Yaskawa INFORM job: R1_W31(0,0)_KM-OK.JBI

/JOB
//NAME R1_W31(0,0)_KM-OK
///FOLDERNAME KRIS-SCIANA
//POS
///NPOS 65,65,0,4,0,0
///TOOL 0
///POSTYPE PULSE
///PULSE
C00000=-3378,-139883,-97046,148601,63097,19554
C00001=-9157,-139883,-97046,148601,63097,19554
C00002=14423,-139883,-97046,148601,63097,19554
C00003=25248,-128582,-94175,152681,55492,17228
C00004=27205,-127666,-93925,153637,54506,16635
C00005=25484,-128476,-94146,152795,55373,17157
C00006=24457,-124392,-93002,151737,54562,17917
C00007=25484,-128476,-94146,152795,55373,17157
C00008=16411,-139658,-96993,149510,62230,18973
C00009=16411,-139658,-96993,149510,62230,18973
C00010=23126,-128454,-94140,151543,56250,17966
C00011=25024,-127329,-93830,152407,55203,17428
C00012=26846,-126477,-93594,153294,54279,16874
C00013=25024,-127329,-93830,152407,55203,17428
C00014=24148,-123758,-92822,151495,54500,18086
C00015=22779,-128284,-94093,151343,56332,18098
C00016=21057,-113910,-69749,152741,63461,16563
C00017=22950,-111460,-69051,153499,62072,16185
C00018=24905,-111066,-68937,154492,61279,15593
C00019=26651,-110455,-68757,155377,60511,15074
C00020=24905,-111066,-68937,154492,61279,15593
C00021=24139,-108709,-68237,153879,60863,16039
C00022=24905,-111066,-68937,154492,61279,15593
C00023=21365,-129655,-79903,153341,64942,15994
C00024=21365,-129655,-79903,153341,64942,15994
C00025=21365,-129655,-79903,153341,64942,15994
C00026=20940,-133487,-97884,150530,57334,18616
C00027=26110,-127410,-97825,152085,52729,17755
///LIMIT ON
C00028=-107604,79582,41685,153491,37881,19627
C00029=-107224,79409,41473,153690,37712,19470
///LIMIT OFF
C00030=26036,-121266,-88084,153104,55194,16958
C00031=22153,-126078,-89436,151612,58043,17810
C00032=26151,-121055,-87868,153174,55168,16910
///LIMIT ON
C00033=-107258,82886,61095,119534,27741,31091
C00034=-106881,82684,60844,119663,27474,31013
///LIMIT OFF
C00035=26195,-120747,-87778,153163,55063,16923
C00036=26195,-120747,-87778,153163,55063,16923
C00037=27152,-120514,-87710,153662,54649,16609
///LIMIT ON
C00038=-107258,82806,60996,119500,27732,31108
C00039=-106881,82604,60746,119629,27464,31030
///LIMIT OFF
C00040=27152,-120514,-87710,153662,54649,16609
C00041=25896,-122880,-88390,153250,55792,16826
C00042=27161,-117906,-83715,154050,55615,16299
C00043=27161,-117906,-83715,154050,55615,16299
///LIMIT ON
C00044=-107257,82726,60897,119467,27722,31125
C00045=-106880,82524,60648,119596,27455,31047
///LIMIT OFF
C00046=27161,-117906,-83715,154050,55615,16299
C00047=26010,-116408,-78989,154106,57886,16118
C00048=26010,-116408,-78989,154106,57886,16118
C00049=27211,-114659,-78882,154502,56737,15929
///LIMIT ON
C00050=-107256,82646,60799,119433,27713,31142
C00051=-106879,82445,60550,119562,27446,31064
///LIMIT OFF
C00052=27209,-114651,-78879,154500,56735,15931
C00053=25407,-114144,-74093,154324,59707,15835
C00054=25407,-110889,-69044,154716,60962,15469
C00055=26831,-107525,-66907,155376,60119,15103
///LIMIT ON
C00056=-107256,82566,60701,119400,27704,31159
C00057=-106879,82365,60452,119529,27437,31081
///LIMIT OFF
C00058=27080,-101000,-56543,156267,62718,14289
C00059=22644,-108994,-60238,154325,65787,15230
C00060=-52788,-93244,-55241,130948,98095,35026
C00061=-80375,-99739,-69495,56806,86442,35710
C00062=-110141,-127728,-104321,3125,87796,34758
C00063=-110141,-127728,-104321,3125,87796,34758
C00064=1472,-127728,-104321,3125,87796,34758
BC00000=204370,1305091,673639
BC00001=2222,1298561,673639
BC00002=2222,1317543,673639
BC00003=2221,1317541,673640
BC00004=2221,1317541,673640
BC00005=2221,1317541,673640
BC00006=2221,1317541,673640
BC00007=2221,1317541,673640
BC00008=2221,1317541,673640
BC00009=2221,1317541,422792
BC00010=2221,1317541,422792
BC00011=2221,1317541,422792
BC00012=2221,1317541,422792
BC00013=2221,1317541,422792
BC00014=2221,1317541,422792
BC00015=2221,1317541,422792
BC00016=2221,1317541,335002
BC00017=2221,1317541,335002
BC00018=2221,1317541,335002
BC00019=2221,1317541,335002
BC00020=2221,1317541,335002
BC00021=2221,1317541,335002
BC00022=2221,1317541,335002
BC00023=2221,1317541,593632
BC00024=2221,1317541,809188
BC00025=12256,1314853,809188
BC00026=2183,1317396,719431
BC00027=2183,1317396,719431
BC00028=39399,1318630,622069
BC00029=39399,1318630,622069
BC00030=2183,1317396,719431
BC00031=2183,1317396,689296
BC00032=2183,1317396,649606
BC00033=22077,1294776,797041
BC00034=22077,1294776,797041
BC00035=2183,1317396,594568
BC00036=1385,1318548,564401
BC00037=2487,1318548,552886
BC00038=22099,1294686,693769
BC00039=22099,1294686,693769
BC00040=2487,1318548,510550
BC00041=2487,1318548,481150
BC00042=2487,1318548,481150
BC00043=2487,1318548,481150
BC00044=22122,1294597,590497
BC00045=22122,1294597,590497
BC00046=2487,1318548,433632
BC00047=2487,1318548,433632
BC00048=2487,1318548,408520
BC00049=2487,1318548,408520
BC00050=22145,1294508,487225
BC00051=22145,1294508,487225
BC00052=2487,1318548,356727
BC00053=2487,1318548,356727
BC00054=2487,1318548,356727
BC00055=2487,1318548,356727
BC00056=22167,1294418,383953
BC00057=22167,1294418,383953
BC00058=2487,1318548,356727
BC00059=2487,1318548,356727
BC00060=2487,1318548,356727
BC00061=3339,1318510,357221
BC00062=22432,1259590,609164
BC00063=22432,703386,940375
BC00064=22432,703386,940375
///POSTYPE BASE
///RECTAN
///RCONF 0,0,0,0,0,0,0,0,0,0,0,0,0,0,0,0,0,0,0,0,0,0,0,0
P00006=0.222,-3.123,-1.508,0.0000,0.0000,0.0000
P00021=-0.225,-6.128,-0.405,0.0000,0.0000,0.0000
P00022=0.222,-3.123,-1.508,0.0000,0.0000,0.0000
P00023=0.143,-0.036,0.682,0.0000,0.0000,0.0000
//INST
///DATE 2024/07/18 18:49
///ATTR SC,RW
///GROUP1 RB1,BS1
NOP
SFTOF
MOVJ C00000 BC00000 VJ=100.00
MOVJ C00001 BC00001 VJ=100.00
MOVL C00002 BC00002 V=333.3
MOVL C00003 BC00003 V=133.3
REFP 3 C00004 BC00004
CALL JOB:SEARCH-R1
SET P021 P006
SFTON P021
MOVL C00005 BC00005 V=133.3
REFP 3 C00006 BC00006
CALL JOB:SEARCH-R1
SET P021 P006
SFTON P021
MOVL C00007 BC00007 V=60.0
SFTOF
MOVJ C00008 BC00008 VJ=50.00
MOVJ C00009 BC00009 VJ=100.00
MOVJ C00010 BC00010 VJ=50.00
MOVL C00011 BC00011 V=133.3
REFP 3 C00012 BC00012
CALL JOB:SEARCH-R1
SET P022 P006
SFTON P022
MOVL C00013 BC00013 V=133.3
REFP 3 C00014 BC00014
CALL JOB:SEARCH-R1
SET P022 P006
SFTON P022
'Path W950
MOVL C00015 BC00015 V=250.0
SFTOF
MOVJ C00016 BC00016 VJ=100.00
MOVL C00017 BC00017 V=400.0
MOVL C00018 BC00018 V=100.0
REFP 3 C00019 BC00019
CALL JOB:SEARCH-R1
SET P023 P006
SFTON P023
MOVL C00020 BC00020 V=133.3
REFP 3 C00021 BC00021
CALL JOB:SEARCH-R1
SET P023 P006
SFTON P023
MOVL C00022 BC00022 V=400.0
SFTOF
MOVJ C00023 BC00023 VJ=100.00
MOVJ C00024 BC00024 VJ=100.00
SFTON P021
MOVJ C00025 BC00025 VJ=100.00
MOVL C00026 BC00026 V=333.3
MOVL C00027 BC00027 V=100.0 PL=0
REFP 1 C00028 BC00028
REFP 2 C00029 BC00029
MACRO1 MJ#(0) ARGF10
ARCON
MOVL C00030 BC00030 V=10.8
ARCOF
MOVL C00031 BC00031 V=250.0
MOVL C00032 BC00032 V=166.7 PL=0
REFP 1 C00033 BC00033
REFP 2 C00034 BC00034
MACRO1 MJ#(0) ARGF10
ARCON
MOVL C00035 BC00035 V=10.8
ARCOF
MOVL C00036 BC00036 V=333.3
MOVL C00037 BC00037 V=166.7 PL=0
REFP 1 C00038 BC00038
REFP 2 C00039 BC00039
ARCON
MOVL C00040 BC00040 V=10.8
ARCOF
MOVL C00041 BC00041 V=250.0
MOVL C00042 BC00042 V=250.0
SFTON P022
MOVL C00043 BC00043 V=250.0 PL=0
REFP 1 C00044 BC00044
REFP 2 C00045 BC00045
ARCON
MOVL C00046 BC00046 V=10.8
ARCOF
MOVL C00047 BC00047 V=250.0
MOVL C00048 BC00048 V=333.3
MOVL C00049 BC00049 V=166.7 PL=0
REFP 1 C00050 BC00050
REFP 2 C00051 BC00051
ARCON
MOVL C00052 BC00052 V=10.8
ARCOF
MOVL C00053 BC00053 V=250.0
SFTOF
MOVL C00054 BC00054 V=333.3
SFTON P023
MOVL C00055 BC00055 V=166.7 PL=0
REFP 1 C00056 BC00056
REFP 2 C00057 BC00057
ARCON
MOVL C00058 BC00058 V=10.8
ARCOF
SFTOF
MOVL C00059 BC00059 V=250.0
MOVJ C00060 BC00060 VJ=50.00
MOVJ C00061 BC00061 VJ=50.00
MOVJ C00062 BC00062 VJ=50.00
SFTOF
MOVJ C00063 BC00063 VJ=100.00
MOVJ C00064 BC00064 VJ=50.00
END
